FUNCTION_BLOCK PCDSMotion
VAR_INPUT
	bEnable: BOOL;
	bInitCfg: BOOL := TRUE;
	bCfgRO: BOOL := FALSE;
	bLimitFwd: BOOL;
	bLimitBwd: BOOL;
	bHomeSensor: BOOL;
	amsEncAddr: AMSADDR;
	nEncCh: USINT;
END_VAR
VAR_IN_OUT
	stConfigSet: ST_AxisParams;
END_VAR
VAR_OUTPUT
	bBrakeOut: BOOL;
	stConfigGet: ST_AxisParams;
END_VAR
VAR
	fbLink: FB_NcAxis;
	fbHardware: FB_AxisHardware;
	fbConfig: FB_AxisConfig;
	fbAxisOP: FB_AxisOP;
	fbDrive: FB_DriveVirtual;
	stAxisStatus: DUT_AxisStatus_v0_01;
	bExecConfig: BOOL;
END_VAR

// Landing zone to link the AXIS_REF and update it
fbLink(En:=bEnable);
// Get terminal info
fbHardware(bExecute:=bEnable,
	Axis:=fbLink.Axis,
	amsEncAddr:=amsEncAddr,
	nEncCh:=nEncCh);
// If asked to initialize and we haven't, then initialize
IF bInitCfg AND NOT fbConfig.bInit THEN
	bExecConfig := TRUE;
// If read-only and not initializing, reject the write command
ELSIF bCfgRO THEN
	bExecConfig := FALSE;
// Otherwise, keep the value written over ADS
END_IF
// Read and/or write the config
fbConfig(bExecute:=bExecConfig AND fbHardware.bDone,
	stConfigSet:=stConfigSet,
	stHardware:=fbHardware.stHardware,
	Axis:=fbLink.Axis,
	stConfigGet=>stConfigGet);
// Reset the execute bool
IF fbConfig.bDone AND NOT fbConfig.bError THEN
	bExecConfig := FALSE;
END_IF
// After the initial config is done, go to OP mode
fbAxisOP(bEnable:=fbConfig.bInit OR NOT bInitCfg,
	stHardware:=fbHardware.stHardware);
// Disable brake while executing move **TODO** make this robust
bBrakeOut := fbDrive.bExecute;
// Execute incoming motion commands
fbDrive(En:=bEnable,
	bEnable:=bEnable AND fbConfig.bInit AND NOT fbConfig.bWriting,
	bLimitFwd:=bLimitFwd,
	bLimitBwd:=bLimitBwd,
	bHomeSensor:=bHomeSensor,
	Axis:=fbLink.Axis);
stAxisStatus := fbDrive.stAxisStatus;
// Reset the execute bool
IF fbDrive.bDone AND NOT fbDrive.bError THEN
	fbDrive.bExecute := FALSE;
END_IF

END_FUNCTION_BLOCK

(* stored: Version 1.1.0.1, ProductVersion 3.1.4020.12
   POU PCDSMotion: Id {ffde42e9-8ab9-4b2d-b01e-b36e19e1042f}, SpecialFunc None *)
